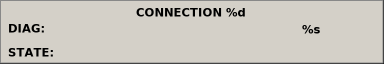
VISUALIZATION V_PH_CONNECTION  // 384x64
VAR_INPUT
		wIndex						: WORD;
		stSafetyStausConnection		:ST_SAFETYStatusConnection;
END_VAR
    Rectangle (0,0 384x64)
    Rectangle (102,1 178x23), "CONNECTION %d", text variable: wIndex
    Rectangle (60,17 232x25), text list: 'TL_ConnectionDiag', text index: stSafetyStausConnection.eSAFETY_ConnectionDiag0F
    Rectangle (299,17 75x25), "%s", text variable: stSafetyStausConnection.sSAFETY_ConnectionDiagF0
    Rectangle (60,38 314x25), text list: 'TL_ConnectionState', text index: stSafetyStausConnection.eSAFETY_ConnectionState
    Label (5,18 43x21), "DIAG:"
    Label (5,38 51x29), "STATE:"
END_VISUALIZATION

(* stored: Version 1.1.0.1, ProductVersion 3.1.4024.4
   Visu V_PH_CONNECTION: Id {ec779b46-acb2-4134-a385-638b44d205de} *)
